Fanuc KAREL source: kt00078.KL

-- PROVISIONAL review KL for V1013-1; original PC SHA256 32b8e57f568de7bb40c2734da81a0d18ad2e834162ec215c32e95d2f2d3c2172
-- Incomplete behavior may be omitted. Consult companion uncertainty JSON. Do not deploy.
PROGRAM KT00078
%NOLOCKGROUP
VAR
  R1 : REAL
  OUT : REAL
-- UNRESOLVED_DECL Y2 type=002018
BEGIN
  -- UNRESOLVED_PC offsets 5-16; opcodes 2E,23
  -- UNRESOLVED_PC offsets 21-35; opcodes 2E,22,9D,33,B2
  -- UNRESOLVED_PC offsets 40-63; opcodes 21,22,9D,33,B1,64,6B,23
  -- UNRESOLVED_PC offsets 68-72; opcodes 7F
END KT00078
